FUNCTION_BLOCK AI_FB_CTUD (* Up-Down counter (INT) AI-Adapter Version *)
  (* Standard: 61499-2; Description: Copyright (c) 2026 Meisterschulen am Ostbahnhof This program and the accompanying materials are made available under the terms of the Eclipse Public License 2.0 which is available at https://www.eclipse.org/legal/epl-2.0/ SPDX-License-Identifier: EPL-2.0 NOTE: This block fires the AX output events (QU.E1, QD.E1, CV.E1, etc.) only on value changes using the internal E_D_FF_* change-driven wiring (e.g., E_D_FF_QU, E_D_FF_QD, E_D_FF_ANY_PV, E_D_FF_CU, E_D_FF_CD, E_D_FF_R, E_D_FF_LD). External filtering is no longer required. *)
  (* Version 1.0, 2026-04-21, Franz Höpfinger, Meisterschulen am Ostbahnhof, initial API and implementation and/or initial documentation *)
  PACKAGE adapter::iec61131::counters;
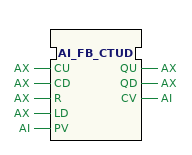
  SOCKETS
    CU : adapter::types::unidirectional::AX; (* Count up *)
    CD : adapter::types::unidirectional::AX; (* Count down *)
    R : adapter::types::unidirectional::AX; (* Reset *)
    LD : adapter::types::unidirectional::AX; (* Load *)
    PV : adapter::types::unidirectional::AI; (* Preset value *)
  END_SOCKETS
  PLUGS
    QU : adapter::types::unidirectional::AX; (* Output Up *)
    QD : adapter::types::unidirectional::AX; (* Output Down *)
    CV : adapter::types::unidirectional::AI; (* Count value *)
  END_PLUGS
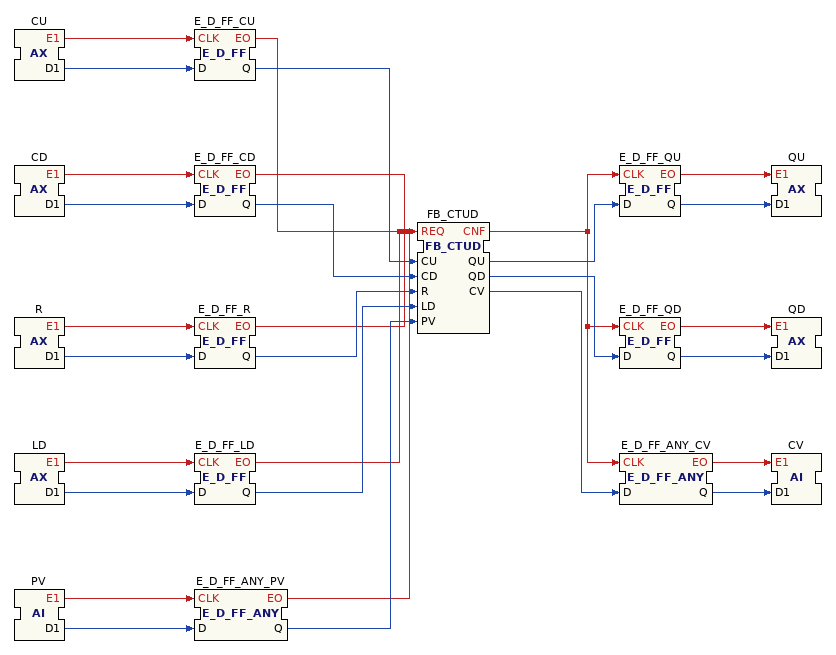
  FBS
    FB_CTUD : iec61131::counters::FB_CTUD;
    E_D_FF_CU : iec61499::events::E_D_FF;
    E_D_FF_CD : iec61499::events::E_D_FF;
    E_D_FF_R : iec61499::events::E_D_FF;
    E_D_FF_LD : iec61499::events::E_D_FF;
    E_D_FF_ANY_PV : iec61499::events::E_D_FF_ANY;
    E_D_FF_QU : iec61499::events::E_D_FF;
    E_D_FF_QD : iec61499::events::E_D_FF;
    E_D_FF_ANY_CV : iec61499::events::E_D_FF_ANY;
  END_FBS
  EVENT_CONNECTIONS
    CU.E1 TO E_D_FF_CU.CLK;
    E_D_FF_CU.EO TO FB_CTUD.REQ;
    CD.E1 TO E_D_FF_CD.CLK;
    E_D_FF_CD.EO TO FB_CTUD.REQ;
    R.E1 TO E_D_FF_R.CLK;
    E_D_FF_R.EO TO FB_CTUD.REQ;
    LD.E1 TO E_D_FF_LD.CLK;
    E_D_FF_LD.EO TO FB_CTUD.REQ;
    PV.E1 TO E_D_FF_ANY_PV.CLK;
    E_D_FF_ANY_PV.EO TO FB_CTUD.REQ;
    FB_CTUD.CNF TO E_D_FF_QU.CLK;
    E_D_FF_QU.EO TO QU.E1;
    FB_CTUD.CNF TO E_D_FF_QD.CLK;
    E_D_FF_QD.EO TO QD.E1;
    FB_CTUD.CNF TO E_D_FF_ANY_CV.CLK;
    E_D_FF_ANY_CV.EO TO CV.E1;
  END_CONNECTIONS
  DATA_CONNECTIONS
    CU.D1 TO E_D_FF_CU.D;
    E_D_FF_CU.Q TO FB_CTUD.CU;
    CD.D1 TO E_D_FF_CD.D;
    E_D_FF_CD.Q TO FB_CTUD.CD;
    R.D1 TO E_D_FF_R.D;
    E_D_FF_R.Q TO FB_CTUD.R;
    LD.D1 TO E_D_FF_LD.D;
    E_D_FF_LD.Q TO FB_CTUD.LD;
    PV.D1 TO E_D_FF_ANY_PV.D;
    E_D_FF_ANY_PV.Q TO FB_CTUD.PV;
    FB_CTUD.QU TO E_D_FF_QU.D;
    E_D_FF_QU.Q TO QU.D1;
    FB_CTUD.QD TO E_D_FF_QD.D;
    E_D_FF_QD.Q TO QD.D1;
    FB_CTUD.CV TO E_D_FF_ANY_CV.D;
    E_D_FF_ANY_CV.Q TO CV.D1;
  END_CONNECTIONS
END_FUNCTION_BLOCK
